FUNCTION_BLOCK FB_System_HS_131
VAR_INPUT
	Freigabe_auto			: BOOL;
	Betrieb_Anford_auto		: BOOL;
	Regelung_Modus_auto		: SINT;
END_VAR
VAR_OUTPUT
	{attribute 'OPC.UA.DA' := '1'}Parameter					: ST_System_HS_Parameter;	
	{attribute 'OPC.UA.DA' := '1'}Steuerung					: ST_System_HS_Steuerung;	
	{attribute 'OPC.UA.DA' := '1'}Zustand						: ST_System_HS_Zustand;	
END_VAR
VAR
	Heizstaebe_131_KW			: FB_HS;
	Regelung					: FB_System_HS_Regelung;
	Zustandscheck				: FB_System_HS_Zustandscheck;
	Logik						: FB_System_HS_Logik;
	Sollwertscheck				: FB_System_HS_Sollwertscheck;
END_VAR

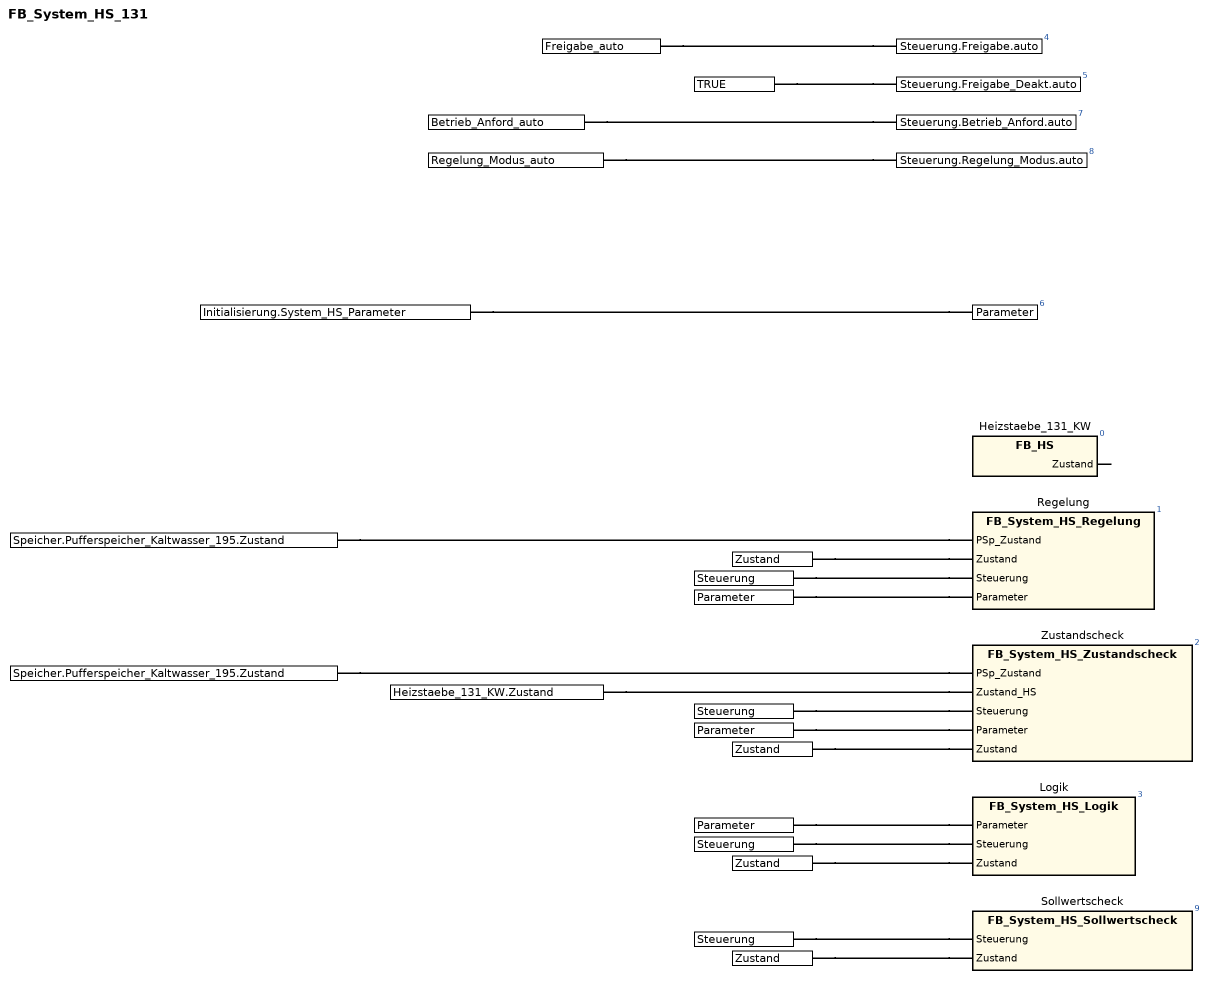
Heizstaebe_131_KW(); // FB_HS
Regelung(
    PSp_Zustand := Speicher.Pufferspeicher_Kaltwasser_195.Zustand,
    Zustand := Zustand,
    Steuerung := Steuerung,
    Parameter := Parameter); // FB_System_HS_Regelung
Zustandscheck(
    PSp_Zustand := Speicher.Pufferspeicher_Kaltwasser_195.Zustand,
    Zustand_HS := Heizstaebe_131_KW.Zustand,
    Steuerung := Steuerung,
    Parameter := Parameter,
    Zustand := Zustand); // FB_System_HS_Zustandscheck
Logik(Parameter := Parameter, Steuerung := Steuerung, Zustand := Zustand); // FB_System_HS_Logik
Steuerung.Freigabe.auto := Freigabe_auto;
Steuerung.Freigabe_Deakt.auto := TRUE;
Parameter := Initialisierung.System_HS_Parameter;
Steuerung.Betrieb_Anford.auto := Betrieb_Anford_auto;
Steuerung.Regelung_Modus.auto := Regelung_Modus_auto;
Sollwertscheck(Steuerung := Steuerung, Zustand := Zustand); // FB_System_HS_Sollwertscheck

END_FUNCTION_BLOCK

(* stored: Version 1.1.0.1, ProductVersion 3.1.4024.9
   POU FB_System_HS_131: Id {2408e43c-6411-4d6f-b0d7-e0b9c7329d70}, SpecialFunc None *)
